FUNCTION_BLOCK FLOTMACHMODEL (* flotation reservoiur *)
  (* Version 1.0, AN, SWDC RTSoft *)
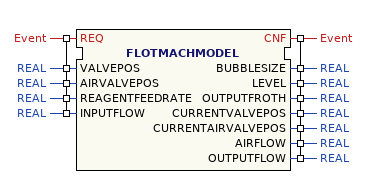
  EVENT_INPUT
    REQ WITH VALVEPOS, AIRVALVEPOS, REAGENTFEEDRATE, INPUTFLOW;
  END_EVENT
  EVENT_OUTPUT
    CNF WITH BUBBLESIZE, LEVEL, OUTPUTFROTH, CURRENTVALVEPOS, CURRENTAIRVALVEPOS, AIRFLOW, OUTPUTFLOW;
  END_EVENT
  VAR_INPUT
    VALVEPOS : REAL;
    AIRVALVEPOS : REAL;
    REAGENTFEEDRATE : REAL;
    INPUTFLOW : REAL;
  END_VAR
  VAR_OUTPUT
    BUBBLESIZE : REAL;
    LEVEL : REAL;
    OUTPUTFROTH : REAL;
    CURRENTVALVEPOS : REAL;
    CURRENTAIRVALVEPOS : REAL;
    AIRFLOW : REAL;
    OUTPUTFLOW : REAL;
  END_VAR
END_FUNCTION_BLOCK
